// TIA Portal V19 export
FUNCTION_BLOCK "OpCycleAnalisys"   // FB1854, LAD
TITLE = Op Cycle analisys
AUTHOR : Piemme
// stored: Access Published, MemoryReserve 100, SetENOAutomatically false
   VAR_INPUT
      CoordinationIn : Struct
         OperationX : Struct
            GoToWork : Bool;
            GoToRest : Bool;
            IsAtWork : Bool;
            IsAtRest : Bool;
            Reset : Bool;
         END_STRUCT;
      END_STRUCT;
   END_VAR
   VAR_IN_OUT
      OperationX_TIME_1 : Time;
      OperationX_TIME_2 : Time;
      OperationX_TIME_3 : Time;
      OperationX_TOTAL : Time;
   END_VAR
   VAR
      Now : Date_And_Time;
      Fp1 : Bool;
      Fp2 : Bool;
      Fp3 : Bool;
      Fp4 : Bool;
      Fp5 : Bool;
      Fp6 : Bool;
      Fp7 : Bool;
      Fp8 : Bool;
      Fp9 : Bool;
      Fp10 : Bool;
      Fp11 : Bool;
      Fp12 : Bool;
      DT_1 : Date_And_Time;
      DT_2 : Date_And_Time;
      DT_3 : Date_And_Time;
   END_VAR
   VAR_TEMP
      RetVal : Int;
   END_VAR
   VAR_TEMP   // added for the SCL form of the ladder/FBD networks
      _w1 : Bool;
      _w2 : Bool;
      _w3 : Bool;
      _w4 : Bool;
      _w5 : Bool;
   END_VAR
BEGIN

REGION Network 1: Now
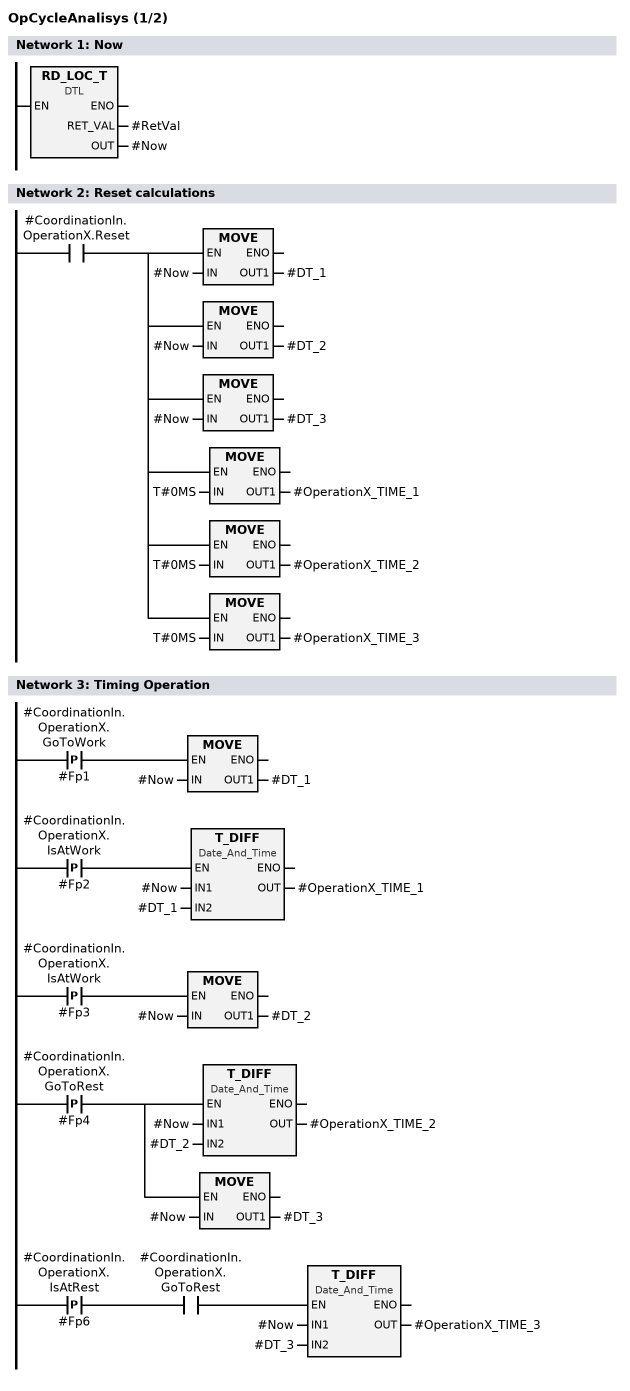
   RUNG wire#powerrail
      { S7_Templates := "date_type := DTL" } RD_LOC_T(RET_VAL => #RetVal, OUT => #Now)
   END_RUNG
   // the same network as SCL:
   #RetVal := RD_LOC_T(OUT => #Now);
END_REGION

REGION Network 2: Reset calculations
   RUNG wire#powerrail
      Contact( #CoordinationIn.OperationX.Reset )
      wire#w1
      Move(in := #Now, out1 => #DT_1)
   END_RUNG
   RUNG wire#w1
      Move(in := #Now, out1 => #DT_2)
   END_RUNG
   RUNG wire#w1
      Move(in := #Now, out1 => #DT_3)
   END_RUNG
   RUNG wire#w1
      { S7_GenerateENO := "TRUE" } Move(in := T#0MS, out1 => #OperationX_TIME_1)
   END_RUNG
   RUNG wire#w1
      { S7_GenerateENO := "TRUE" } Move(in := T#0MS, out1 => #OperationX_TIME_2)
   END_RUNG
   RUNG wire#w1
      { S7_GenerateENO := "TRUE" } Move(in := T#0MS, out1 => #OperationX_TIME_3)
   END_RUNG
   // the same network as SCL:
   IF #CoordinationIn.OperationX.Reset THEN
       #DT_1 := #Now;
       #DT_2 := #Now;
       #DT_3 := #Now;
       #OperationX_TIME_1 := T#0MS;
       #OperationX_TIME_2 := T#0MS;
       #OperationX_TIME_3 := T#0MS;
   END_IF;
END_REGION

REGION Network 3: Timing Operation
   RUNG wire#powerrail
      P_Contact(operand := #CoordinationIn.OperationX.GoToWork, bit := #Fp1)
      Move(in := #Now, out1 => #DT_1)
   END_RUNG
   RUNG wire#powerrail
      P_Contact(operand := #CoordinationIn.OperationX.IsAtWork, bit := #Fp2)
      { S7_Templates := "[date_type := Date_And_Time, time_type := Time]" } T_DIFF(IN1 := #Now, IN2 := #DT_1, OUT => #OperationX_TIME_1)
   END_RUNG
   RUNG wire#powerrail
      P_Contact(operand := #CoordinationIn.OperationX.IsAtWork, bit := #Fp3)
      Move(in := #Now, out1 => #DT_2)
   END_RUNG
   RUNG wire#powerrail
      P_Contact(operand := #CoordinationIn.OperationX.GoToRest, bit := #Fp4)
      wire#w1
      { S7_Templates := "[date_type := Date_And_Time, time_type := Time]" } T_DIFF(IN1 := #Now, IN2 := #DT_2, OUT => #OperationX_TIME_2)
   END_RUNG
   RUNG wire#w1
      Move(in := #Now, out1 => #DT_3)
   END_RUNG
   RUNG wire#powerrail
      P_Contact(operand := #CoordinationIn.OperationX.IsAtRest, bit := #Fp6)
      Contact( #CoordinationIn.OperationX.GoToRest )
      { S7_Templates := "[date_type := Date_And_Time, time_type := Time]" } T_DIFF(IN1 := #Now, IN2 := #DT_3, OUT => #OperationX_TIME_3)
   END_RUNG
   // the same network as SCL:
   #_w1 := #CoordinationIn.OperationX.GoToWork AND NOT #Fp1;   // rising edge of #CoordinationIn.OperationX.GoToWork
   #Fp1 := #CoordinationIn.OperationX.GoToWork;
   IF #_w1 THEN #DT_1 := #Now; END_IF;
   #_w2 := #CoordinationIn.OperationX.IsAtWork AND NOT #Fp2;   // rising edge of #CoordinationIn.OperationX.IsAtWork
   #Fp2 := #CoordinationIn.OperationX.IsAtWork;
   IF #_w2 THEN T_DIFF(IN1 := #Now, IN2 := #DT_1, OUT => #OperationX_TIME_1); END_IF;
   #_w3 := #CoordinationIn.OperationX.IsAtWork AND NOT #Fp3;   // rising edge of #CoordinationIn.OperationX.IsAtWork
   #Fp3 := #CoordinationIn.OperationX.IsAtWork;
   IF #_w3 THEN #DT_2 := #Now; END_IF;
   #_w4 := #CoordinationIn.OperationX.GoToRest AND NOT #Fp4;   // rising edge of #CoordinationIn.OperationX.GoToRest
   #Fp4 := #CoordinationIn.OperationX.GoToRest;
   IF #_w4 THEN
       T_DIFF(IN1 := #Now, IN2 := #DT_2, OUT => #OperationX_TIME_2);
       #DT_3 := #Now;
   END_IF;
   #_w5 := #CoordinationIn.OperationX.IsAtRest AND NOT #Fp6;   // rising edge of #CoordinationIn.OperationX.IsAtRest
   #Fp6 := #CoordinationIn.OperationX.IsAtRest;
   IF #_w5 AND #CoordinationIn.OperationX.GoToRest THEN
       T_DIFF(IN1 := #Now, IN2 := #DT_3, OUT => #OperationX_TIME_3);
   END_IF;
END_REGION

REGION Network 4: Total time calculation
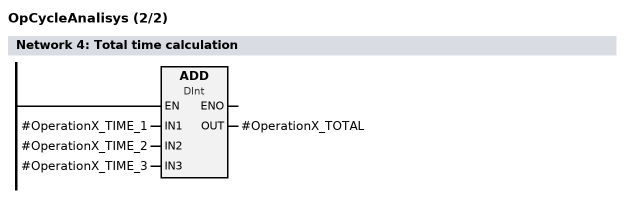
   RUNG wire#powerrail
      { S7_Templates := "SrcType := DInt"; S7_GenerateENO := "TRUE" } Add(in1 := #OperationX_TIME_1, in2 := #OperationX_TIME_2, in3 := #OperationX_TIME_3, out => #OperationX_TOTAL)
   END_RUNG
   // the same network as SCL:
   #OperationX_TOTAL := #OperationX_TIME_1 + #OperationX_TIME_2 + #OperationX_TIME_3;
END_REGION
END_FUNCTION_BLOCK
